TYPE ST_MOVER_SELECTOR_CTRL :
STRUCT
  Selector      : E_MOVER_SELECTOR; // select by array Index OR AXIS_REF.NcToPlc.AxisId 
  Mover         : UINT;             // array Index OR AXIS_REF.NcToPlc.AxisId
  Control       : ST_MOVER_CTRL;    // mover control struct, put motion command in here

  Data          : ST_MOVE_DATA;     // write your movement parameters
  //Gear          : ST_GEAR_DATA;     // write your gearing parameters
END_STRUCT
END_TYPE

(* stored: Version 1.1.0.1, ProductVersion 3.1.4026.20
   DUT ST_MOVER_SELECTOR_CTRL: Id {5c2f5d54-f475-44a3-acc1-8f761e3b080e} *)
